// TwinCAT 3 PLC project PLC_ST02
// ProgramVersion: 3.1.4024.0
// libraries:
//   Base Objects Library, * (JABIL RAC LATAM)
//   Tc2_MC2, * (Beckhoff Automation GmbH)
//   Tc2_Standard, * (Beckhoff Automation GmbH)
//   Tc2_System, * (Beckhoff Automation GmbH)
//   Tc3_Module, * (Beckhoff Automation GmbH)
// project tree:
//   / PlcST02Task.TcTTO
//   POUs/00-MainPRG/ MAIN_ST02.TcPOU
//   POUs/02-FunctionBlocks/TanslationStation/ FB_TranslationStation.TcPOU
//   POUs/02-FunctionBlocks/Tapping/ EN_TapeInSystemStatus.TcDUT, FB_TapeAplicationMahine.TcPOU, FB_TapeApplicator.TcPOU
// (motion and I/O tree: see PLC project plc_st01)
// real-time tasks:
//   TASK PlcST01Task: cycle T#10ms, priority 20, ADS port 350
//   TASK PlcST02Task: cycle T#10ms, priority 21, ADS port 351
//   TASK PlcST03Task: cycle T#10ms, priority 22, ADS port 352
// variable links:

CONFIGURATION PLC_ST02
    RESOURCE PLC ON TwinCAT3
        TASK PlcST02Task(INTERVAL := T#10ms, PRIORITY := 21);
        PROGRAM MAIN_ST02 WITH PlcST02Task : MAIN_ST02;
    END_RESOURCE
END_CONFIGURATION

// ---- POUs/02-FunctionBlocks/Tapping/EN_TapeInSystemStatus.TcDUT
{attribute 'qualified_only'}
{attribute 'strict'}
{attribute 'to_string'}
TYPE EN_TapeInSystemStatus :
(
	tapeOnlyInPickPlate,
	tapeGrippedInPicker,
	tapeCutted,
	tapeOnApplyPlates
);
END_TYPE

// ---- POUs/00-MainPRG/MAIN_ST02.TcPOU
PROGRAM MAIN_ST02
VAR
	fbStation02							: RACBaseObjects.FB_Station;
	fbTranslationStationIn				: FB_TranslationStation;
	fbConveyor							: RACBaseObjects.FB_Conveyor;
	fbTapeApplicationMachine			: FB_TapeAplicationMahine;
	fbTranslationStationOut				: FB_TranslationStation;
END_VAR

	fbStation02(						bInitFinished := fbTapeApplicationMachine.bInit_Finished);

	fbTranslationStationIn(				sDeviceID := '', 
										bStopExecution := fbStation02.bStop,
										bAlarmReset := fbStation02.bAlarmReset,
										diStationState := fbStation02.diStationState,
										bInit_StartPermissive := FALSE);

	fbConveyor(							sDeviceID := '', 
										bStopExecution := fbStation02.bStop,
										bAlarmReset := fbStation02.bAlarmReset,
										diStationState := fbStation02.diStationState,
										bInit_StartPermissive := FALSE);

	fbTapeApplicationMachine(
										sDeviceID := '', 
										bStopExecution := fbStation02.bStop,
										bAlarmReset := fbStation02.bAlarmReset,
										diStationState := fbStation02.diStationState,
										bInit_StartPermissive := FALSE);

	fbTranslationStationOut(			sDeviceID := '', 
										bStopExecution := fbStation02.bStop,
										bAlarmReset := fbStation02.bAlarmReset,
										diStationState := fbStation02.diStationState,
										bInit_StartPermissive := FALSE);

END_PROGRAM

// ---- POUs/02-FunctionBlocks/TanslationStation/FB_TranslationStation.TcPOU
FUNCTION_BLOCK FB_TranslationStation EXTENDS RACBaseObjects.FB_Machine
VAR_INPUT
	sRobotID						: STRING;
	
	sRejectCartID					: STRING;
	sLockCylinerID					: STRING;
	
	bSafetyBoxPick_permissive		: BOOL;
	bPick_OKPieceReady				: BOOL;
	bPick_NGPieceReady				: BOOL;
	
	bSafetyBoxPlace_permisive		: BOOL;
	bPlace_ReadyToRecieve			: BOOL;
END_VAR
VAR_OUTPUT
	bSafetyBoxPick_outOfZone		: BOOL;
	bPick_done						: BOOL;
	
	bSafetyBoxPlace_outOfZone		: BOOL;
	bPlace_done						: BOOL;
END_VAR
VAR
	fbRobot							: RACBaseObjects.FB_Robot;
	fbRejectCart					: RACBaseObjects.FB_RejectCart;
END_VAR

//	Run the standar main for any machine
SUPER^.MachineMain();

//	Robot instance
	fbRobot(							sDeviceID:=	sRobotID,
										bStopExecution:=bStopExecution,
										bAlarmReset:=bAlarmReset,
										diStationState:=diStationState,
										bInit_StartPermissive:=bInit_StartPermissive,
										bSafetyBoxPick_Permissive:=bSafetyBoxPick_permissive,
										bSafetyBoxPlace_Permissive:=bSafetyBoxPlace_permisive,
										bSafetyBoxReject_Permissive:=fbRejectCart.bSafetyBox_okForEnter,
										bOKMaterialReadyToPick:=bPick_OKPieceReady,
										bNGMaterialReadyToPick:=bPick_NGPieceReady,
										bPiceIsGood:=TRUE,
										bPiceIsNG:=FALSE,
										bPlace_MaterialRequest:=bPlace_ReadyToRecieve,
										bReject_MaterialRequest:=FALSE,
										bSafetyBoxPick_OutOfZone=>bSafetyBoxPick_outOfZone,
										bSafetyBoxPlace_OutOfZone=>bSafetyBoxPlace_outOfZone,
										bPick_AllMaterialPicked=>bPick_done,
										bPlace_Done=>bPlace_Done);

//	Reject cart instance
	fbRejectCart(						sDeviceID:=	sRejectCartID,
										bStopExecution:=bStopExecution,
										bAlarmReset:=bAlarmReset,
										diStationState:=diStationState,
										bInit_StartPermissive:=fbRobot.bInit_Finished,
										sLockCylinerID:=sLockCylinerID,
										bSafetyBox_permissive:=fbRobot.bSafetyBoxReject_OutOfZone,
										bPlacePieceOnCartRequest:=);

METHOD  Alarm
sAlarm									:= CONCAT (STR1:=fbRobot.sAlarm,STR2:=fbRejectCart.sAlarm);
END_METHOD

METHOD  Auto
END_METHOD

METHOD  Init
bInit_Finished							:= fbRobot.bInit_Finished and fbRejectCart.bInit_Finished;
END_METHOD

METHOD  IO
END_METHOD

METHOD  Manual
END_METHOD

METHOD  Pause
END_METHOD

METHOD  Stop
END_METHOD

END_FUNCTION_BLOCK

// ---- POUs/02-FunctionBlocks/Tapping/FB_TapeAplicationMahine.TcPOU
FUNCTION_BLOCK FB_TapeAplicationMahine EXTENDS RACBaseObjects.FB_Machine
VAR_INPUT
END_VAR
VAR_OUTPUT
END_VAR
VAR
	fbServo_Translational						: RACBaseObjects.FB_Motor;
	fbTapeApplicator_Left						: FB_TapeApplicator;
	fbTapeApplicator_Right						: FB_TapeApplicator;
END_VAR

SUPER^.MachineMain();

//	Both tape applicator systems traslation servo
	fbServo_Translational(		sDeviceID:='',
								bStopExecution:=bStopExecution,
								bAlarmReset:=bAlarmReset,
								diStationState:=diStationState,
								bInit_StartPermissive:=(fbTapeApplicator_Left.bAllServosSafePosition AND fbTapeApplicator_Right.bAllServosSafePosition),
								bMovePermissive:=(fbTapeApplicator_Left.bSafeConditions AND fbTapeApplicator_Right.bSafeConditions));

//	Left tape applicator system
	fbTapeApplicator_Left(		sDeviceID:='',
								bStopExecution:=bStopExecution,
								bAlarmReset:=bAlarmReset,
								diStationState:=diStationState,
								bInit_StartPermissive:=bInit_StartPermissive,
								sSvoLiftID:='',
								sSvoPickrID:='',
								sCylScissorsID:='',
								sCylTapeAppFrontID:='',
								sCylTapeAppRearID:='',
								sCylVaccID:='',
								sCylPickerID:='');

//	Right tape applicator system
	fbTapeApplicator_Right(		sDeviceID:='',
								bStopExecution:=bStopExecution,
								bAlarmReset:=bAlarmReset,
								diStationState:=diStationState,
								bInit_StartPermissive:=bInit_StartPermissive,
								sSvoLiftID:='',
								sSvoPickrID:='',
								sCylScissorsID:='',
								sCylTapeAppFrontID:='',
								sCylTapeAppRearID:='',
								sCylVaccID:='',
								sCylPickerID:='');

METHOD Alarm
sAlarm:= CONCAT(STR1:=fbServo_Translational.sAlarm, STR2:=fbTapeApplicator_Left.sAlarm);
sAlarm:= CONCAT(STR1:=sAlarm,STR2:=fbTapeApplicator_Right.sAlarm);
END_METHOD

METHOD Auto
END_METHOD

METHOD Init
bInit_Finished:= (fbServo_Translational.bInit_Finished AND fbTapeApplicator_Left.bInit_Finished AND fbTapeApplicator_Right.bInit_Finished);
END_METHOD

METHOD IO
END_METHOD

METHOD Manual
END_METHOD

METHOD Pause
END_METHOD

METHOD Stop
END_METHOD

END_FUNCTION_BLOCK

// ---- POUs/02-FunctionBlocks/Tapping/FB_TapeApplicator.TcPOU
FUNCTION_BLOCK FB_TapeApplicator EXTENDS RACBaseObjects.FB_Machine
VAR_INPUT
	sSvoLiftID								: STRING;
	sSvoPickrID								: STRING;
	sCylScissorsID							: STRING;
	sCylTapeAppFrontID						: STRING;
	sCylTapeAppRearID						: STRING;
	sCylVaccID								: STRING;
	sCylPickerID							: STRING;
	sVaccPickPlateID						: STRING;
	sVaccFrontPlateID						: STRING;
	sVaccRearPlateID						: STRING;
END_VAR
VAR_OUTPUT
	bSafeConditions							: BOOL							:=FALSE;
	
	bAllServosSafePosition					: BOOL							:=FALSE;
	bAllCylinderSafePosition				: BOOL							:=FALSE;
END_VAR
VAR
	bServo_Lift_isSafePosition				: BOOL							:=FALSE;
	bServo_Picker_isSafePosition			: BOOL							:=FALSE;
	
	bTapeInPicker							AT%I* : BOOL;
		
	tapeInSystemStatus						: EN_TapeInSystemStatus			:=EN_TapeInSystemStatus.tapeOnlyInPickPlate;

	fbServo_Lift							: RACBaseObjects.FB_Motor;
	fbServo_Picker							: RACBaseObjects.FB_Motor;
	
	fbCyl_Scissors							: RACBaseObjects.FB_Cylinder;
	fbCyl_TapeApplicatorFront				: RACBaseObjects.FB_Cylinder;
	fbCyl_TapeApplicatorRear				: RACBaseObjects.FB_Cylinder;
	fbCyl_Vacc								: RACBaseObjects.FB_Cylinder;
	fbCyl_Picker							: RACBaseObjects.FB_Cylinder;
	
	fbVacc_PickPlate						: RACBaseObjects.FB_Vacuum;
	fbVacc_FrontPlate						: RACBaseObjects.FB_Vacuum;
	fbVacc_RearPlate						: RACBaseObjects.FB_Vacuum;
END_VAR

SUPER^.MachineMain();

//	Lift tape applicator
	fbServo_Lift(				sDeviceID:=sSvoLiftID,
								bStopExecution:=bStopExecution,
								bAlarmReset:=bAlarmReset,
								diStationState:=diStationState,
								bInit_StartPermissive:=fbCyl_TapeApplicatorFront.bIsRetracted AND fbCyl_TapeApplicatorRear.bIsRetracted,
								bMovePermissive:=bServo_Picker_isSafePosition AND fbCyl_TapeApplicatorFront.bIsRetracted AND fbCyl_TapeApplicatorRear.bIsRetracted);
	bServo_Lift_isSafePosition		:= (fbServo_Lift.lrActualPosition<=20) OR (fbServo_Lift.lrActualPosition>=100);

//	Move tape picker rear - front						
	fbServo_Picker(				sDeviceID:=sSvoPickrID,
								bStopExecution:=bStopExecution,
								bAlarmReset:=bAlarmReset,
								diStationState:=diStationState,
								bInit_StartPermissive:=fbServo_Lift.bInit_Finished,
								bMovePermissive:=bServo_Lift_isSafePosition);
	bServo_Picker_isSafePosition	:= (fbServo_Picker.lrActualPosition<=100);

//	Scissors Cylinder
	fbCyl_Scissors(				sDeviceID:=sCylScissorsID,
								bStopExecution:=bStopExecution,
								bAlarmReset:=bAlarmReset,
								bPermisiveExtend:=TRUE,
								bPermisiveRetract:=TRUE,
								Timeout:=T#1S);

//	Tape applicator frontal Cylinder
	fbCyl_TapeApplicatorFront(	sDeviceID:=sCylTapeAppFrontID,
								bStopExecution:=bStopExecution,
								bAlarmReset:=bAlarmReset,
								bPermisiveExtend:=bServo_Lift_isSafePosition,
								bPermisiveRetract:=TRUE,
								Timeout:=T#1S);

//	Tape applicator rear Cylinder
	fbCyl_TapeApplicatorRear(	sDeviceID:=sCylTapeAppRearID,
								bStopExecution:=bStopExecution,
								bAlarmReset:=bAlarmReset,
								bPermisiveExtend:=bServo_Lift_isSafePosition,
								bPermisiveRetract:=TRUE,
								Timeout:=T#1S);

//	Vacc Cylinder
	fbCyl_Vacc(					sDeviceID:=sCylVaccID,
								bStopExecution:=bStopExecution,
								bAlarmReset:=bAlarmReset,
								bPermisiveExtend:=bServo_Picker_isSafePosition,
								bPermisiveRetract:=bServo_Picker_isSafePosition,
								Timeout:=T#1S);

//	Picker Cylinder
	fbCyl_Picker(				sDeviceID:=sCylPickerID,
								bStopExecution:=bStopExecution,
								bAlarmReset:=bAlarmReset,
								bPermisiveExtend:=TRUE,
								bPermisiveRetract:=TRUE,
								Timeout:=T#1S);

//	Pick Plate Vaccum Generator
	fbVacc_PickPlate(			sDeviceID:=sVaccPickPlateID,
								bStopExecution:=bStopExecution,
								bAlarmReset:=bAlarmReset,
								Timeout:=T#1S);

//	Front Plate Vaccum Generator
	fbVacc_FrontPlate(			sDeviceID:=sVaccFrontPlateID,
								bStopExecution:=bStopExecution,
								bAlarmReset:=bAlarmReset,
								Timeout:=T#1S);

//	Rear Plate Vaccum Generator
	fbVacc_FrontPlate(			sDeviceID:=sVaccRearPlateID,
								bStopExecution:=bStopExecution,
								bAlarmReset:=bAlarmReset,
								Timeout:=T#1S);

METHOD Alarm
sAlarm:= CONCAT(STR1:=fbServo_Lift.sAlarm,STR2:=fbServo_Picker.sAlarm);
sAlarm:= CONCAT(STR1:=sAlarm,STR2:=fbCyl_Scissors.sAlarm);
sAlarm:= CONCAT(STR1:=sAlarm,STR2:=fbCyl_TapeApplicatorFront.sAlarm);
sAlarm:= CONCAT(STR1:=sAlarm,STR2:=fbCyl_TapeApplicatorRear.sAlarm);
sAlarm:= CONCAT(STR1:=sAlarm,STR2:=fbCyl_Vacc.sAlarm);
sAlarm:= CONCAT(STR1:=sAlarm,STR2:=fbCyl_Picker.sAlarm);
sAlarm:= CONCAT(STR1:=sAlarm,STR2:=fbVacc_PickPlate.sAlarm);
sAlarm:= CONCAT(STR1:=sAlarm,STR2:=fbVacc_FrontPlate.sAlarm);
sAlarm:= CONCAT(STR1:=sAlarm,STR2:=fbVacc_RearPlate.sAlarm);
END_METHOD

METHOD Auto
//	Keep sequencer in range
	IF (diActualSeqStep<1000) OR (diActualSeqStep>1999) THEN
		diActualSeqStep:=1000;
	END_IF

//	Automatic sequence
	CASE diActualSeqStep OF
		1000:	//	Evaluate status of tape in system
		1001:	//	Validate tape is on vacc supported in pick plate
		1010:	//	Open picker cylinder
		1020:	//	Move pick servo to tape pick position
		1030:	//	Close picker cylinder
		1040:	//	Move pick servo to tape release postion
		1050:	//	Turn ON Vacc in front and rear plate
		1060:	//	Open picker cylinder
		1070:	//	
		1099:	//	Turn OFF vacc in rear and front plate, retract rear plate cylinder and move lift servo to safe position
	END_CASE
END_METHOD

METHOD Init
//	Keep sequencer in range
	IF (diActualSeqStep<0) OR (diActualSeqStep>999) THEN
		diActualSeqStep:=0;
	END_IF

//	Initialization sequence
	CASE diActualSeqStep OF
		0:		//	Wait init start permissive
			IF bInit_StartPermissive THEN
				diActualSeqStep								:=	10;
			END_IF
		10:		//	Turn ON pick plate vaccum generator and validate feedback
			IF NOT fbVacc_PickPlate.bGrip THEN
				fbVacc_PickPlate.bGrip						:=	TRUE;
			END_IF
			IF fbVacc_PickPlate.Vacuum_Ok THEN
				diActualSeqStep								:=	20;
			END_IF
		20:		//	Update tape in system status
			IF fbCyl_Picker.bIsRetracted AND bTapeInPicker THEN
				tapeInSystemStatus						:=	EN_TapeInSystemStatus.tapeGrippedInPicker;
			END_IF
			IF (tapeInSystemStatus=EN_TapeInSystemStatus.tapeGrippedInPicker) AND fbCyl_Scissors.bIsRetracted THEN
				tapeInSystemStatus						:=	EN_TapeInSystemStatus.tapeCutted;
			END_IF
			IF (tapeInSystemStatus=EN_TapeInSystemStatus.tapeGrippedInPicker) AND fbCyl_Scissors.bIsRetracted THEN
				tapeInSystemStatus						:=	EN_TapeInSystemStatus.tapeOnApplyPlates;
			END_IF
			diActualSeqStep								:=	30;
		30:		//	Set cylincer in safe position to init servos
			fbCyl_TapeApplicatorFront.bRetractRequest	:=	(NOT fbCyl_TapeApplicatorFront.bIsRetracted);
			fbCyl_TapeApplicatorRear.bRetractRequest	:=	(NOT fbCyl_TapeApplicatorRear.bIsRetracted);
			fbCyl_Vacc.bRetractRequest					:=	(NOT fbCyl_Vacc.bIsRetracted);
			IF fbCyl_Scissors.bIsExtended AND fbCyl_TapeApplicatorFront.bIsRetracted AND fbCyl_TapeApplicatorRear.bIsRetracted AND fbCyl_Vacc.bIsRetracted THEN 
				diActualSeqStep							:=	30;
			END_IF
		40:		//	Wait servos init finished
			IF fbServo_Lift.bInit_Finished AND fbServo_Picker.bInit_Finished THEN
				diActualSeqStep							:=	40;
			END_IF
		50:		//	Set scissors cylinder open
			fbCyl_Scissors.bExtendRequest				:=	NOT fbCyl_Scissors.bIsExtended;
			IF fbCyl_Scissors.bIsExtended THEN 
				diActualSeqStep							:=	60;
			END_IF
		100:	//	Validate pick plate vaccum
			bInit_Finished								:= fbVacc_PickPlate.Vacuum_Ok;
			IF bInit_Finished THEN
				diActualSeqStep							:=	999;
			END_IF
	END_CASE
END_METHOD

METHOD IO
bAllServosSafePosition						:=	bServo_Lift_isSafePosition AND bServo_Picker_isSafePosition;
bAllCylinderSafePosition					:=	fbCyl_TapeApplicatorFront.bIsRetracted AND fbCyl_TapeApplicatorRear.bIsRetracted AND fbCyl_Vacc.bIsRetracted;
bSafeConditions								:=	bAllServosSafePosition AND bAllCylinderSafePosition;
END_METHOD

METHOD Manual
END_METHOD

METHOD Pause
END_METHOD

METHOD Stop
END_METHOD

END_FUNCTION_BLOCK
